_CFC_ (* Continuous Function Chart, elements in execution order *)
(* 3s *)
(* 3s *)
(* 90s *)
(* 1s *)
#0 AND(#3.Q, #6.Q)
#1 INT_TO_TIME(SCHU_P2_2_ZADER_VPDS_OTSUT)
#2 MUL(#1, 1000)
#3 TON_PDS2:TON(IN: NOT SCHU_P2_2_PDS2_DI2, PT: #2)
#4 INT_TO_TIME(SCHU_P2_2_ZADER_VPDS_RABOTA)
#5 MUL(#4, 1000)
#6 TON_ReRab:TON(IN: SCHU_P2_2_UST_RE_RABOTA, PT: #5)
#7 INT_TO_TIME(SCHU_P2_2_ZADER_M_VKL)
#8 MUL(#7, 1000)
#9 TON_MVKL_M1:TON(IN: SCHU_P2_2_SA1_DO1, PT: #8)
#10 INT_TO_TIME(SCHU_P2_2_ZADER_M_A)
#11 MUL(#10, 1000)
#12 TON_AVT_M1:TON(IN: SCHU_P2_2_SA1_DI5_A, PT: #11)
#13 AND(#0, SCHU_P2_2_M1_B30, #9.Q, #12.Q)
#14 SR_NP_M1:SR(SET1: #13, RESET: SCHU_P2_2_SB)
#15 AND(#14.Q1, #18.Q1)
#16 SCHU_P2_2_Z_NetP <= #15
#17 AND(#0, SCHU_P2_2_M2_B30, #21.Q, #24.Q)
#18 SR_NP_M2:SR(SET1: #17, RESET: SCHU_P2_2_SB)
#19 INT_TO_TIME(SCHU_P2_2_ZADER_M_VKL)
#20 MUL(#19, 1000)
#21 TON_MVKL_M2:TON(IN: SCHU_P2_2_SA8_DO8, PT: #20)
#22 INT_TO_TIME(SCHU_P2_2_ZADER_M_A)
#23 MUL(#22, 1000)
#24 TON_AVT_M2:TON(IN: SCHU_P2_2_SA8_DI3_A, PT: #23)
#25 SCHU_P2_2_Z_NetP_M1 <= #14.Q1
#26 SCHU_P2_2_Z_NetP_M2 <= #18.Q1
_END_CFC_
(* the same logic as Structured Text *)
(* 3s *)
(* 3s *)
(* 90s *)
(* 1s *)
_t70 := TON_PDS2.Q AND TON_ReRab.Q;
TON_PDS2(IN := NOT SCHU_P2_2_PDS2_DI2, PT := INT_TO_TIME(SCHU_P2_2_ZADER_VPDS_OTSUT) * 1000);
TON_ReRab(IN := SCHU_P2_2_UST_RE_RABOTA, PT := INT_TO_TIME(SCHU_P2_2_ZADER_VPDS_RABOTA) * 1000);
TON_MVKL_M1(IN := SCHU_P2_2_SA1_DO1, PT := INT_TO_TIME(SCHU_P2_2_ZADER_M_VKL) * 1000);
TON_AVT_M1(IN := SCHU_P2_2_SA1_DI5_A, PT := INT_TO_TIME(SCHU_P2_2_ZADER_M_A) * 1000);
SR_NP_M1(SET1 := _t70 AND SCHU_P2_2_M1_B30 AND TON_MVKL_M1.Q AND TON_AVT_M1.Q, RESET := SCHU_P2_2_SB);
SCHU_P2_2_Z_NetP := SR_NP_M1.Q1 AND SR_NP_M2.Q1;
SR_NP_M2(SET1 := _t70 AND SCHU_P2_2_M2_B30 AND TON_MVKL_M2.Q AND TON_AVT_M2.Q, RESET := SCHU_P2_2_SB);
TON_MVKL_M2(IN := SCHU_P2_2_SA8_DO8, PT := INT_TO_TIME(SCHU_P2_2_ZADER_M_VKL) * 1000);
TON_AVT_M2(IN := SCHU_P2_2_SA8_DI3_A, PT := INT_TO_TIME(SCHU_P2_2_ZADER_M_A) * 1000);
SCHU_P2_2_Z_NetP_M1 := SR_NP_M1.Q1;
SCHU_P2_2_Z_NetP_M2 := SR_NP_M2.Q1;
END_PROGRAM

(* POU TZBiS/TZB/Z_OTKAZ_VTOR_ZEP, CFC *)
PROGRAM Z_OTKAZ_VTOR_ZEP
VAR
	rs_otkaz_vtor_sep: RS;
END_VAR
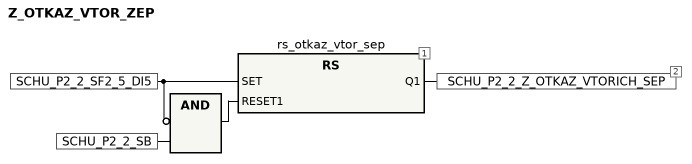
_CFC_ (* Continuous Function Chart, elements in execution order *)
#0 AND(NOT SCHU_P2_2_SF2_5_DI5, SCHU_P2_2_SB)
#1 rs_otkaz_vtor_sep:RS(SET: SCHU_P2_2_SF2_5_DI5, RESET1: #0)
#2 SCHU_P2_2_Z_OTKAZ_VTORICH_SEP <= #1.Q1
_END_CFC_
(* the same logic as Structured Text *)
rs_otkaz_vtor_sep(SET := SCHU_P2_2_SF2_5_DI5, RESET1 := NOT SCHU_P2_2_SF2_5_DI5 AND SCHU_P2_2_SB);
SCHU_P2_2_Z_OTKAZ_VTORICH_SEP := rs_otkaz_vtor_sep.Q1;
END_PROGRAM

(* POU TZBiS/TZB/Z_P1_NP, CFC *)
PROGRAM Z_P1_NP
VAR
	SR_P1_NPit: SR;
END_VAR
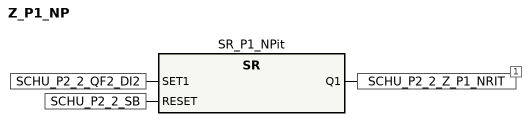
_CFC_ (* Continuous Function Chart, elements in execution order *)
#0 SR_P1_NPit:SR(SET1: SCHU_P2_2_QF2_DI2, RESET: SCHU_P2_2_SB)
#1 SCHU_P2_2_Z_P1_NRIT <= #0.Q1
_END_CFC_
(* the same logic as Structured Text *)
SR_P1_NPit(SET1 := SCHU_P2_2_QF2_DI2, RESET := SCHU_P2_2_SB);
SCHU_P2_2_Z_P1_NRIT := SR_P1_NPit.Q1;
END_PROGRAM

(* POU TZBiS/TZB/Z_P2_NP, CFC *)
PROGRAM Z_P2_NP
VAR
	SR_P2_NPit: SR;
END_VAR
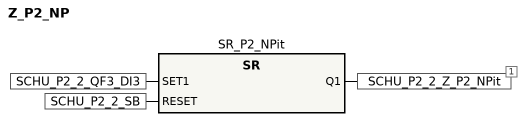
_CFC_ (* Continuous Function Chart, elements in execution order *)
#0 SR_P2_NPit:SR(SET1: SCHU_P2_2_QF3_DI3, RESET: SCHU_P2_2_SB)
#1 SCHU_P2_2_Z_P2_NPit <= #0.Q1
_END_CFC_
(* the same logic as Structured Text *)
SR_P2_NPit(SET1 := SCHU_P2_2_QF3_DI3, RESET := SCHU_P2_2_SB);
SCHU_P2_2_Z_P2_NPit := SR_P2_NPit.Q1;
END_PROGRAM

(* POU TZBiS/TZB/Z_P2_Otk, CFC *)
PROGRAM Z_P2_Otk
VAR
	SR_P2_Otkaz: SR;
	UE2_VL_Old: REAL;
	TON_UE2: TON;
	RT_P2_RUN: R_TRIG;
END_VAR
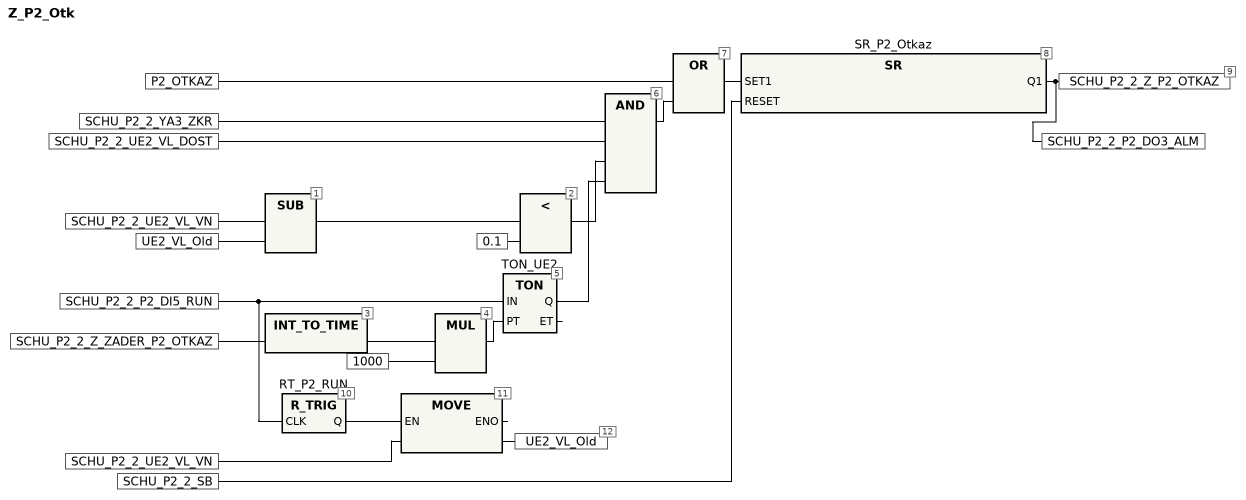
_CFC_ (* Continuous Function Chart, elements in execution order *)
#0 SCHU_P2_2_P2_DO3_ALM <= #8.Q1
#1 SUB(SCHU_P2_2_UE2_VL_VN, UE2_VL_Old)
#2 <(#1, 0.1)
#3 INT_TO_TIME(SCHU_P2_2_Z_ZADER_P2_OTKAZ)
#4 MUL(#3, 1000)
#5 TON_UE2:TON(IN: SCHU_P2_2_P2_DI5_RUN, PT: #4)
#6 AND(SCHU_P2_2_YA3_ZKR, SCHU_P2_2_UE2_VL_DOST, #2, #5.Q)
#7 OR(P2_OTKAZ, #6)
#8 SR_P2_Otkaz:SR(SET1: #7, RESET: SCHU_P2_2_SB)
#9 SCHU_P2_2_Z_P2_OTKAZ <= #8.Q1
#10 RT_P2_RUN:R_TRIG(CLK: SCHU_P2_2_P2_DI5_RUN)
#11 MOVE(EN: #10.Q, SCHU_P2_2_UE2_VL_VN)
#12 UE2_VL_Old <= #11
_END_CFC_
END_PROGRAM

(* POU TZBiS/TZB/Sbros_All, CFC *)
PROGRAM Sbros_All
VAR
END_VAR
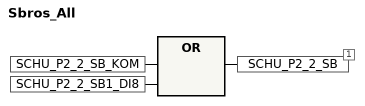
_CFC_ (* Continuous Function Chart, elements in execution order *)
#0 OR(SCHU_P2_2_SB_KOM, SCHU_P2_2_SB1_DI8)
#1 SCHU_P2_2_SB <= #0
_END_CFC_
(* the same logic as Structured Text *)
SCHU_P2_2_SB := SCHU_P2_2_SB_KOM OR SCHU_P2_2_SB1_DI8;
END_PROGRAM

(* POU TZBiS/TZB/Z_Pozhar, CFC *)
PROGRAM Z_Pozhar
VAR
	SR_Pozhar: SR;
END_VAR
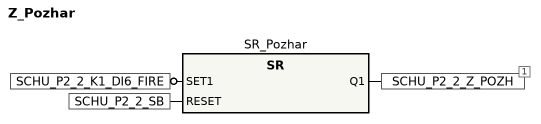
_CFC_ (* Continuous Function Chart, elements in execution order *)
#0 SR_Pozhar:SR(SET1: NOT SCHU_P2_2_K1_DI6_FIRE, RESET: SCHU_P2_2_SB)
#1 SCHU_P2_2_Z_POZH <= #0.Q1
_END_CFC_
(* the same logic as Structured Text *)
SR_Pozhar(SET1 := NOT SCHU_P2_2_K1_DI6_FIRE, RESET := SCHU_P2_2_SB);
SCHU_P2_2_Z_POZH := SR_Pozhar.Q1;
END_PROGRAM

(* POU TZBiS/TZB/Z_YA1_Otk, CFC *)
PROGRAM Z_YA1_Otk
VAR
	SR_YA1_Otkaz: SR;
	TON_YA1_Otk: TON;
	TON_YA1_N_OTKR: TON;
	TON_YA1_N_ZAKR: TON;
	TON_YA1_ZKR: TON;
	TON_AVT: TON;

	a: BOOL;
	b: BOOL;
	c: BOOL;
	d: BOOL;
	e: BOOL;
END_VAR
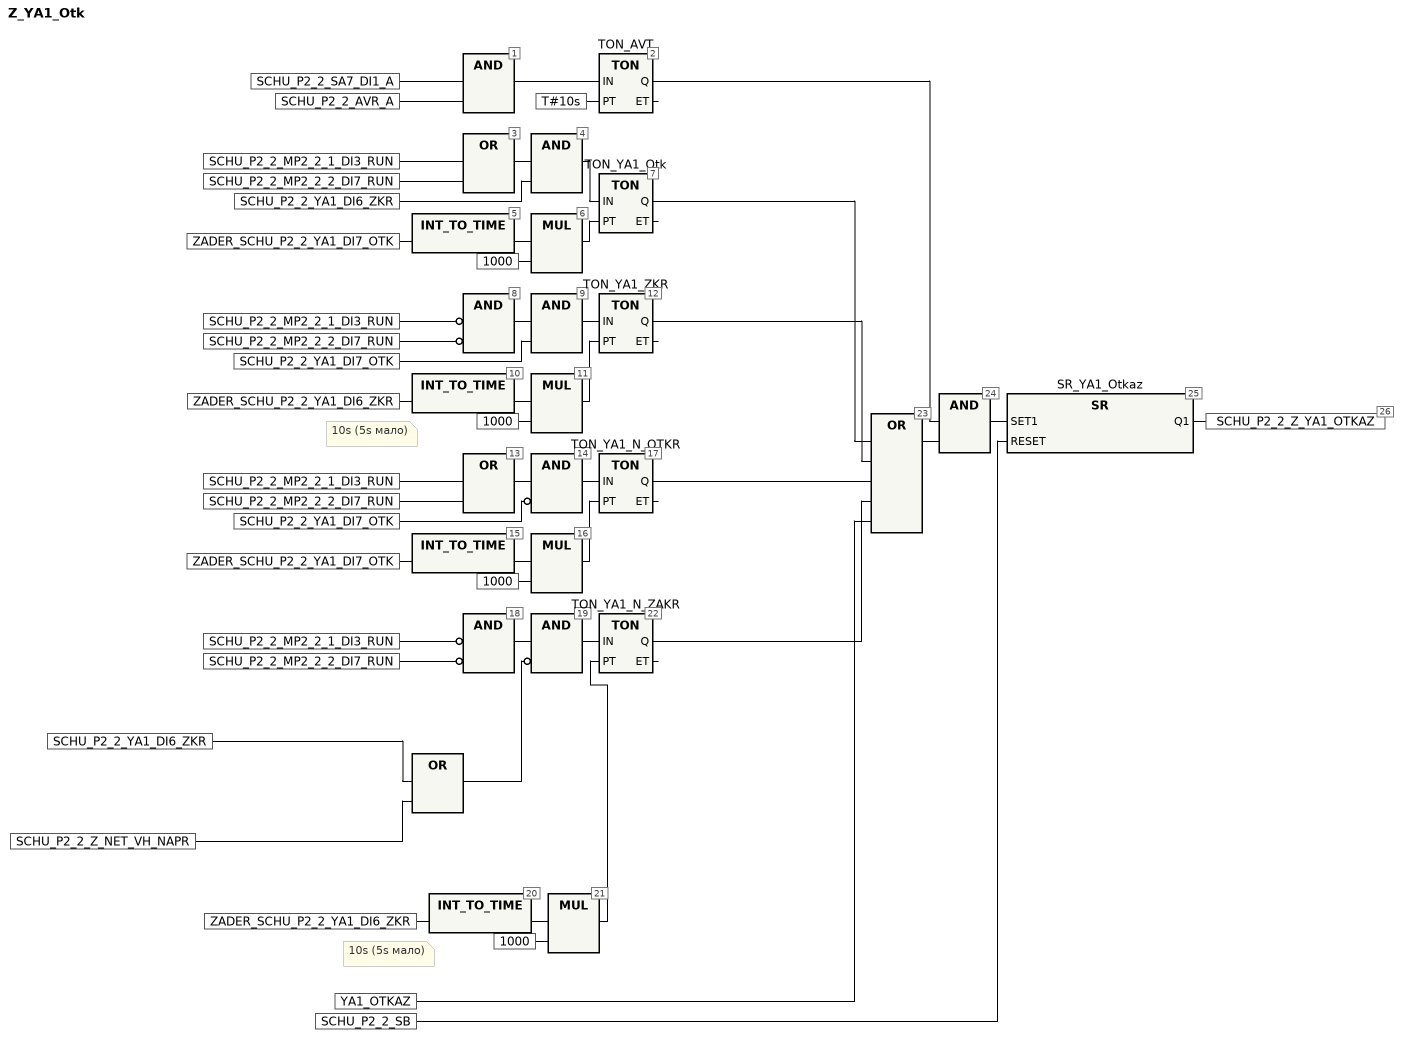
